Omron CX-Programmer project NewProject (CX-Programmer 9.73)

# PLC NewPLC1: CP1L M

## Global symbols (name address type ; comment)
0.00 BOOL  ; Start
0.01 BOOL  ; Close
100.00 BOOL  ; Return to Home
100.01 BOOL  ; Transfer to Conveyor
100.04 BOOL  ; Lower Arm
100.05 BOOL  ; Gripper Close
100.06 BOOL  ; Conveyor
101.00 BOOL  ; Relay
101.11 BOOL  ; Relay

## Program NewProgram1 (cyclic task 0)

### Section Section1

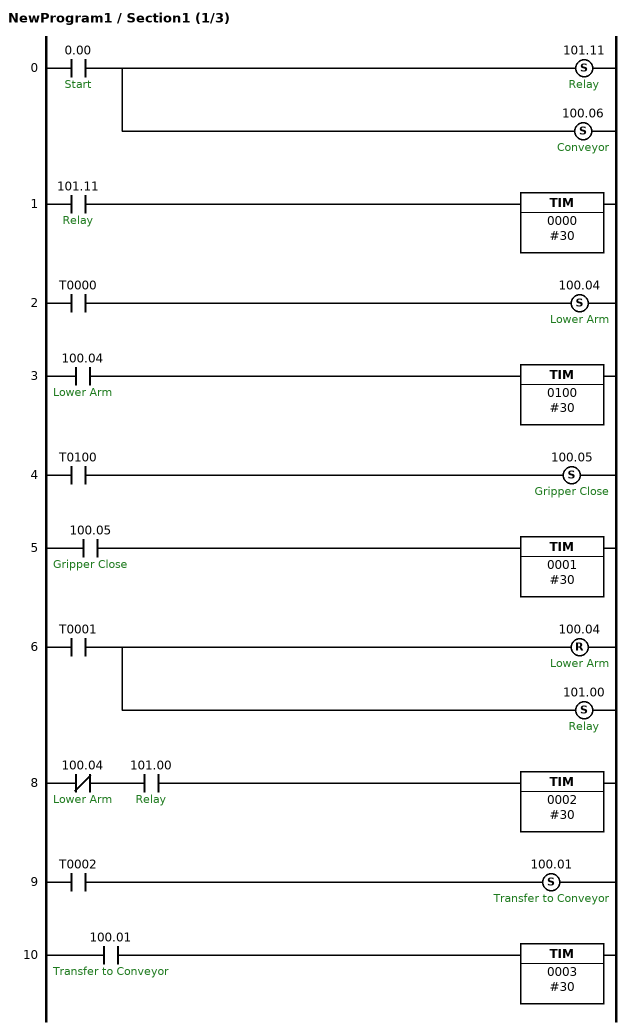
; rung 0
LD 0.00  ; Start
SET 101.11  ; Relay
SET 100.06  ; Conveyor
; rung 1
LD 101.11  ; Relay
TIM 0000 #30
; rung 2
LD T0000
SET 100.04  ; Lower Arm
; rung 3
LD 100.04  ; Lower Arm
TIM 0100 #30
; rung 4
LD T0100
SET 100.05  ; Gripper Close
; rung 5
LD 100.05  ; Gripper Close
TIM 0001 #30
; rung 6
LD T0001
RSET 100.04  ; Lower Arm
SET 101.00  ; Relay
; rung 8
LDNOT 100.04  ; Lower Arm
AND 101.00  ; Relay
TIM 0002 #30
; rung 9
LD T0002
SET 100.01  ; Transfer to Conveyor
; rung 10
LD 100.01  ; Transfer to Conveyor
TIM 0003 #30

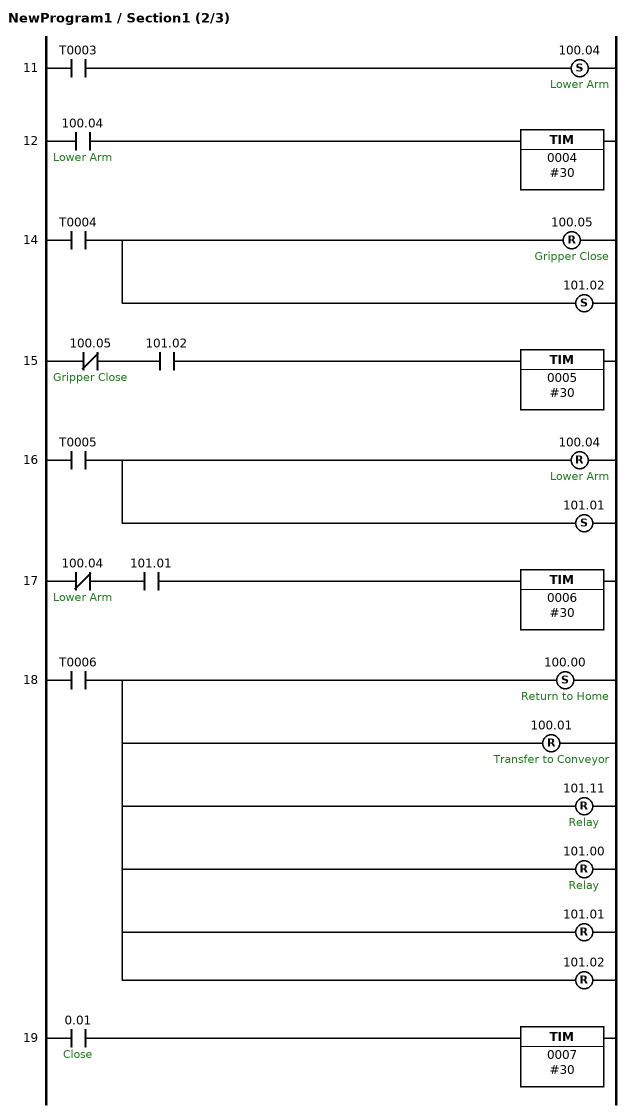
; rung 11
LD T0003
SET 100.04  ; Lower Arm
; rung 12
LD 100.04  ; Lower Arm
TIM 0004 #30
; rung 14
LD T0004
RSET 100.05  ; Gripper Close
SET 101.02
; rung 15
LDNOT 100.05  ; Gripper Close
AND 101.02
TIM 0005 #30
; rung 16
LD T0005
RSET 100.04  ; Lower Arm
SET 101.01
; rung 17
LDNOT 100.04  ; Lower Arm
AND 101.01
TIM 0006 #30
; rung 18
LD T0006
SET 100.00  ; Return to Home
RSET 100.01  ; Transfer to Conveyor
RSET 101.11  ; Relay
RSET 101.00  ; Relay
RSET 101.01
RSET 101.02
; rung 19
LD 0.01  ; Close
TIM 0007 #30

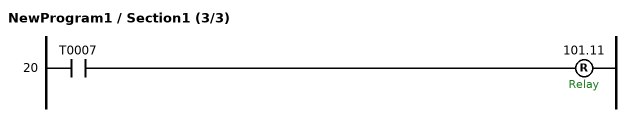
; rung 20
LD T0007
RSET 101.11  ; Relay

### Section END
; rung 0
END(001)